(* Schneider Machine Expert - Basic project M221-KSB-single-pump, file version 2.0.0.0 *)
(* ProjectInformations: Name=KSB Single Pump Panel *)

HARDWARE
  Cpu 0: TM221CE24R
  ModuleExtensionObject 0: TM3TI4/G
  ModuleExtensionObject 1: TM3TI8T/G
  ModuleExtensionObject 2: TM3AI2H/G
  EthernetConfiguration: NetworkName=M221, IpAllocationMode=FixedAddress, IpAddress=192.168.1.107, SubnetMask=255.255.255.0
  SerialLineConfiguration: Baud=Baud19200, Parity=ParityEven, DataBits=DataBits8, StopBits=StopBits1, PhysicalMedium=PhysicalMediumRs485, TransmissionMode=TransmissionModeModbusRtu, SlaveId=1, Addressing=SlaveAddressing
  MastTask: UsePeriodScanMode=false, PeriodScan=100
  FastTask: Period=255
  CpuBehavior: StartingMode=StartInRun, AutoSaveRamOnEeprom=true, WatchdogPeriod=250

SYMBOLS  (address, symbol, comment, settings)
  %M0       SET_PLC_TIME  "Setting this bit allows you to change the PLC Time; gets set on negative transition of bit"
  %M1       SEAL_FAIL_ALARM
  %M2       HIGH_FLOAT_ALARM
  %M3       HIGH_VIBRATION_ALARM
  %M4       HIGH_BOTTOM_BEARING_TEMP_ALARM
  %M5       RESET_ALARMS
  %M6       SILENCE_ALARMS
  %M7       WINDING_TEMP_ALARM_BYPASS
  %M8       SEAL_FAIL_ALARM_BYPASS
  %M9       HIGH_FLOAT_ALARM_BYPASS
  %M10      VIBRATION_ALARM_BYPASS
  %M11      HIGH_BOT_BEAR_TMP_ALARM_BYPASS
  %M12      MODULE_1_STATUS
  %M13      MODULE_2_STATUS
  %M14      MODULE_3_STATUS
  %M110     LOGGING_DONE
  %M111     LOGGING_BUSY
  %M112     LOGGING_ERROR
  %M113     LOGGING_BAK
  %M114     LOG_NEXT
  %S6       SB_TB1S  "Time base of 1 s generated by an internal clock"
  %S13      SB_FIRSTRUN  "Indicates the first controller cycle in RUN mode"
  %S50      SB_RTCUPDATE  "Set to 1, this bit allows to update the date and time"
  %SW51     SW_RTCHHMM  "RTC Function: contains in BCD HHMM: hour and minute"
  %SW52     SW_RTCMMDD  "RTC Function: contains in BCD MMDD: month and day"
  %SW53     SW_RTCCCYY  "RTC Function: contains in BCD CCYY: century and year"
  %SW120    SW_IOSTATUS  "Shows expansion I/O module status (refer F1 help for details)"
  %MW0      DAY
  %MW1      HOUR  "My_Time"
  %MW2      MINUTES
  %MW3      MONTH
  %MW4      YEAR
  %MW5      SCRAP_MONTH  "Interim Register to Load into BCD"
  %MW6      SCRAP_MINUTES  "Interim Register to Load into BCD"
  %MW7      SEAL_FAIL_ALARM_DELAY_PRESET
  %MW8      VIBRATION_ALARM_DELAY_PRESET
  %MW9      WINDING1_TEMP_LOG
  %MW10     WINDING2_TEMP_LOG
  %MW11     WINDING3_TEMP_LOG
  %MW12     BOTTOM_BEARING_TEMP_LOG
  %MW13     WINDING_TEMP_LOG
  %MW14     VIBRATION_LOG
  %KW0      DISCONNECTED_VALUE  [Value=-32768]
  %TM0      HIGH_BOT_BEARING_TMP_ALARM_DELAY  [Preset=10, Base=OneSecond]
  %TM1      HIGH_FLOAT_ALARM_DELAY  [Preset=10, Base=OneSecond]
  %TM2      HIGH_WINDING_TEMP_ALARM_DELAY  [Preset=10, Base=OneSecond]
  %TM3      SEAL_FAIL_ALARM_DELAY  [Preset=10, Base=OneSecond]
  %TM4      VIBRATION_ALARM_DELAY  [Preset=10, Base=OneSecond]
  %TM5      NEXT_LOG_DELAY_TIMER  [Preset=30, Base=OneSecond]
  %DATALOG0   [Records(DataLoggingRecord(Value=%I0.0), DataLoggingRecord(Value=%IW1.0), DataLoggingRecord(Value=%IW1.1), DataLoggingRecord(Value=%IW1.2), DataLoggingRecord(Value=%IW1.3), DataLoggingRecord(Value=%IW2.0), DataLoggingRecord(Value=%IW3.0)), AddDateTime=true, DataLoggingType=HistoricalData, MaxFileSize=100]
  %DATALOG1   [Records(DataLoggingRecord(Value=%IW1.0)), AddDateTime=true, DataLoggingType=HistoricalData, MaxFileSize=500]
  %I0.0     SEAL_FAIL  "Reversed Logic Sensor!!! Normally Closed. Seal failing breaks connection"
  %I0.1     HIGH_FLOAT
  %Q0.0     PUMP_ENABLE
  %Q0.1     AUDIBLE_ALARM
  %IW1.0    WINDING1_TEMP  [Type=Type_PT100, Scope=Scope_Fahrenheit, Minimum=-3280, Maximum=15620]
  %IW1.1    WINDING2_TEMP  [Type=Type_PT100, Scope=Scope_Fahrenheit, Minimum=-3280, Maximum=15620]
  %IW1.2    WINDING3_TEMP  [Type=Type_PT100, Scope=Scope_Fahrenheit, Minimum=-3280, Maximum=15620]
  %IW1.3    BOTTOM_BEARING_TEMP  [Type=Type_PT100, Scope=Scope_Fahrenheit, Minimum=-3280, Maximum=15620]
  %IW2.0    WINDING_TEMP  [Type=Type_NTC, Scope=Scope_Fahrenheit, Minimum=-514, Maximum=1104]
  %IW3.0    VIBRATION  [Type=Type_4_20mA, Scope=Scope_Customized, Minimum=0, Maximum=10000]

POU Alarm Conditions
  (* SectionNumber=1 *)

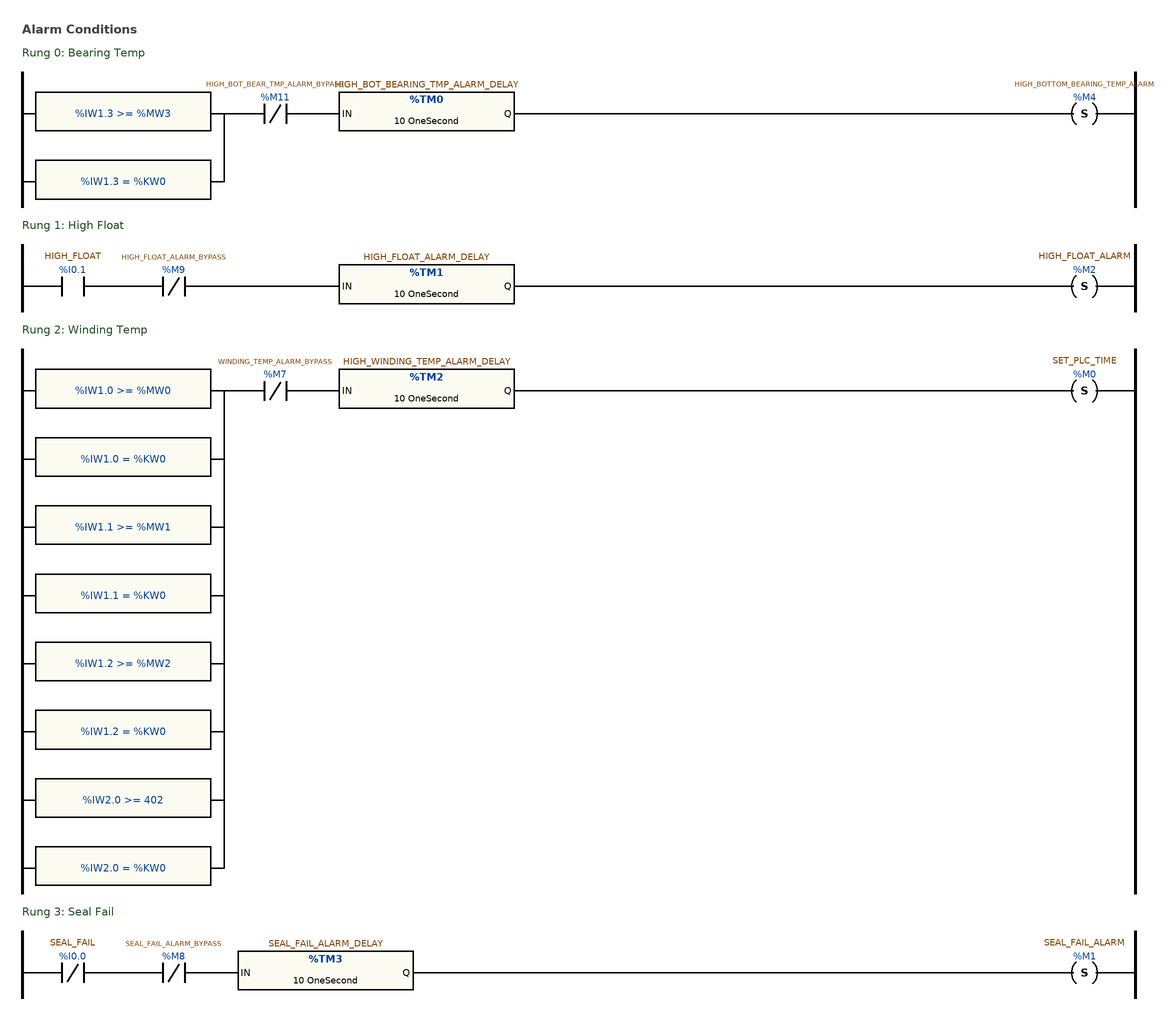

// Rung 0: Bearing Temp
  BLK %TM0                (* HIGH_BOT_BEARING_TMP_ALARM_DELAY *)
  LD [ %IW1.3 >= %MW3 ]   (* BOTTOM_BEARING_TEMP, MONTH *)
  OR [ %IW1.3 = %KW0 ]    (* BOTTOM_BEARING_TEMP, DISCONNECTED_VALUE *)
  ANDN %M11               (* HIGH_BOT_BEAR_TMP_ALARM_BYPASS *)
  IN
  OUT_BLK
  LD Q
  S %M4                   (* HIGH_BOTTOM_BEARING_TEMP_ALARM *)
  END_BLK
  // as ST:
  //   HIGH_BOT_BEARING_TMP_ALARM_DELAY(IN := (BOTTOM_BEARING_TEMP >= MONTH OR BOTTOM_BEARING_TEMP = DISCONNECTED_VALUE) AND NOT HIGH_BOT_BEAR_TMP_ALARM_BYPASS);
  //   IF HIGH_BOT_BEARING_TMP_ALARM_DELAY.Q THEN HIGH_BOTTOM_BEARING_TEMP_ALARM := TRUE; END_IF;

// Rung 1: High Float
  BLK %TM1                (* HIGH_FLOAT_ALARM_DELAY *)
  LD %I0.1                (* HIGH_FLOAT *)
  ANDN %M9                (* HIGH_FLOAT_ALARM_BYPASS *)
  IN
  OUT_BLK
  LD Q
  S %M2                   (* HIGH_FLOAT_ALARM *)
  END_BLK
  // as ST:
  //   HIGH_FLOAT_ALARM_DELAY(IN := HIGH_FLOAT AND NOT HIGH_FLOAT_ALARM_BYPASS);
  //   IF HIGH_FLOAT_ALARM_DELAY.Q THEN HIGH_FLOAT_ALARM := TRUE; END_IF;

// Rung 2: Winding Temp
  BLK %TM2                (* HIGH_WINDING_TEMP_ALARM_DELAY *)
  LD [ %IW1.0 >= %MW0 ]   (* WINDING1_TEMP, DAY *)
  OR [ %IW1.0 = %KW0 ]    (* WINDING1_TEMP, DISCONNECTED_VALUE *)
  OR [ %IW1.1 >= %MW1 ]   (* WINDING2_TEMP, HOUR *)
  OR [ %IW1.1 = %KW0 ]    (* WINDING2_TEMP, DISCONNECTED_VALUE *)
  OR [ %IW1.2 >= %MW2 ]   (* WINDING3_TEMP, MINUTES *)
  OR [ %IW1.2 = %KW0 ]    (* WINDING3_TEMP, DISCONNECTED_VALUE *)
  OR [ %IW2.0 >= 402 ]    (* WINDING_TEMP *)
  OR [ %IW2.0 = %KW0 ]    (* WINDING_TEMP, DISCONNECTED_VALUE *)
  ANDN %M7                (* WINDING_TEMP_ALARM_BYPASS *)
  IN
  OUT_BLK
  LD Q
  S %M0                   (* SET_PLC_TIME *)
  END_BLK
  // as ST:
  //   HIGH_WINDING_TEMP_ALARM_DELAY(IN := (WINDING1_TEMP >= DAY OR WINDING1_TEMP = DISCONNECTED_VALUE OR WINDING2_TEMP >= HOUR OR WINDING2_TEMP = DISCONNECTED_VALUE OR WINDING3_TEMP >= MINUTES OR WINDING3_TEMP = DISCONNECTED_VALUE OR WINDING_TEMP >= 402 OR WINDING_TEMP = DISCONNECTED_VALUE) AND NOT WINDING_TEMP_ALARM_BYPASS);
  //   IF HIGH_WINDING_TEMP_ALARM_DELAY.Q THEN SET_PLC_TIME := TRUE; END_IF;

// Rung 3: Seal Fail
  BLK %TM3                (* SEAL_FAIL_ALARM_DELAY *)
  LDN %I0.0               (* SEAL_FAIL *)
  ANDN %M8                (* SEAL_FAIL_ALARM_BYPASS *)
  IN
  OUT_BLK
  LD Q
  S %M1                   (* SEAL_FAIL_ALARM *)
  END_BLK
  // as ST:
  //   SEAL_FAIL_ALARM_DELAY(IN := NOT SEAL_FAIL AND NOT SEAL_FAIL_ALARM_BYPASS);
  //   IF SEAL_FAIL_ALARM_DELAY.Q THEN SEAL_FAIL_ALARM := TRUE; END_IF;

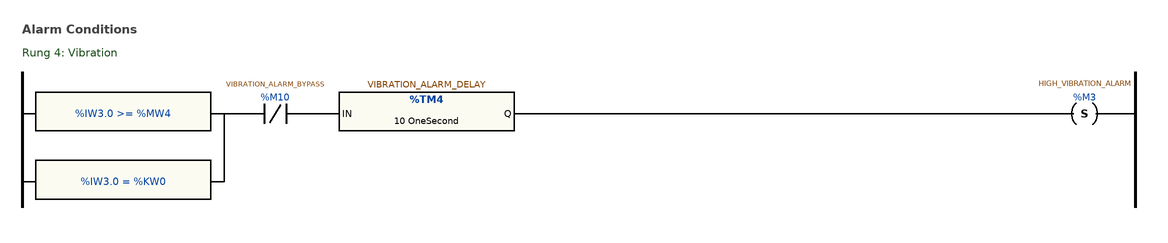

// Rung 4: Vibration
  BLK %TM4                (* VIBRATION_ALARM_DELAY *)
  LD [ %IW3.0 >= %MW4 ]   (* VIBRATION, YEAR *)
  OR [ %IW3.0 = %KW0 ]    (* VIBRATION, DISCONNECTED_VALUE *)
  ANDN %M10               (* VIBRATION_ALARM_BYPASS *)
  IN
  OUT_BLK
  LD Q
  S %M3                   (* HIGH_VIBRATION_ALARM *)
  END_BLK
  // as ST:
  //   VIBRATION_ALARM_DELAY(IN := (VIBRATION >= YEAR OR VIBRATION = DISCONNECTED_VALUE) AND NOT VIBRATION_ALARM_BYPASS);
  //   IF VIBRATION_ALARM_DELAY.Q THEN HIGH_VIBRATION_ALARM := TRUE; END_IF;

POU Pump Enable
  (* SectionNumber=2 *)

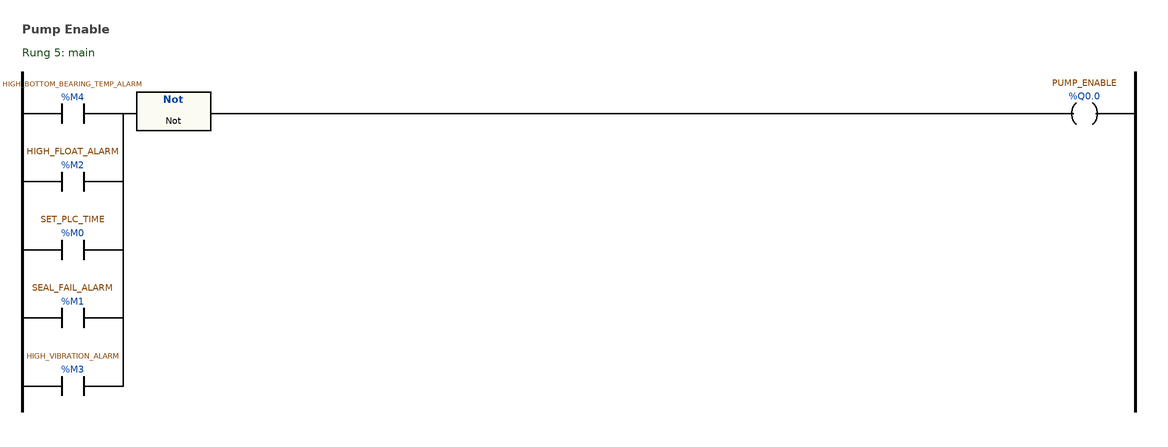

// Rung 5: main
  LD %M4                  (* HIGH_BOTTOM_BEARING_TEMP_ALARM *)
  OR %M2                  (* HIGH_FLOAT_ALARM *)
  OR %M0                  (* SET_PLC_TIME *)
  OR %M1                  (* SEAL_FAIL_ALARM *)
  OR %M3                  (* HIGH_VIBRATION_ALARM *)
  N
  ST %Q0.0                (* PUMP_ENABLE *)
  // as ST:
  //   PUMP_ENABLE := NOT (HIGH_BOTTOM_BEARING_TEMP_ALARM OR HIGH_FLOAT_ALARM OR SET_PLC_TIME OR SEAL_FAIL_ALARM OR HIGH_VIBRATION_ALARM);

POU Resets
  (* SectionNumber=3 *)

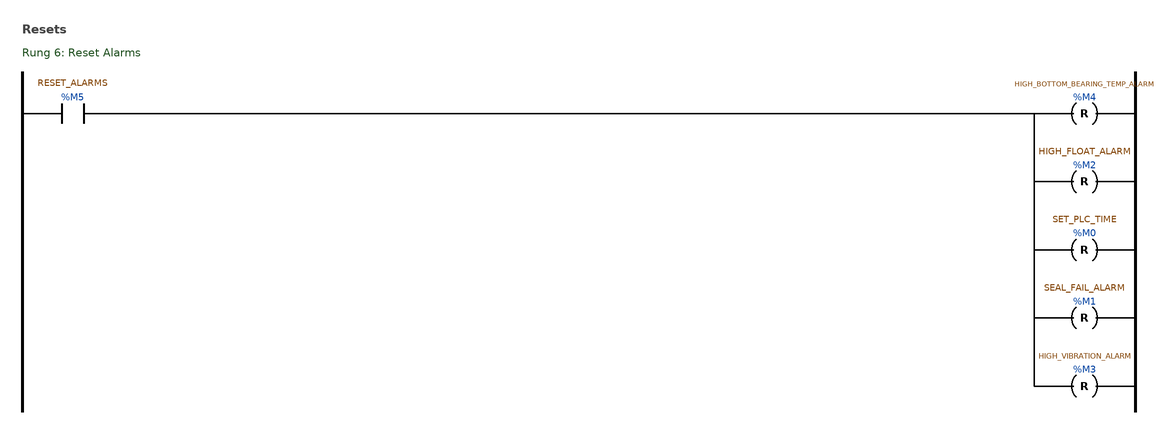

// Rung 6: Reset Alarms
  LD %M5                  (* RESET_ALARMS *)
  R %M4                   (* HIGH_BOTTOM_BEARING_TEMP_ALARM *)
  R %M2                   (* HIGH_FLOAT_ALARM *)
  R %M0                   (* SET_PLC_TIME *)
  R %M1                   (* SEAL_FAIL_ALARM *)
  R %M3                   (* HIGH_VIBRATION_ALARM *)
  // as ST:
  //   IF RESET_ALARMS THEN HIGH_BOTTOM_BEARING_TEMP_ALARM := FALSE; END_IF;
  //   IF RESET_ALARMS THEN HIGH_FLOAT_ALARM := FALSE; END_IF;
  //   IF RESET_ALARMS THEN SET_PLC_TIME := FALSE; END_IF;
  //   IF RESET_ALARMS THEN SEAL_FAIL_ALARM := FALSE; END_IF;
  //   IF RESET_ALARMS THEN HIGH_VIBRATION_ALARM := FALSE; END_IF;

POU On Startup
  (* SectionNumber=4 *)

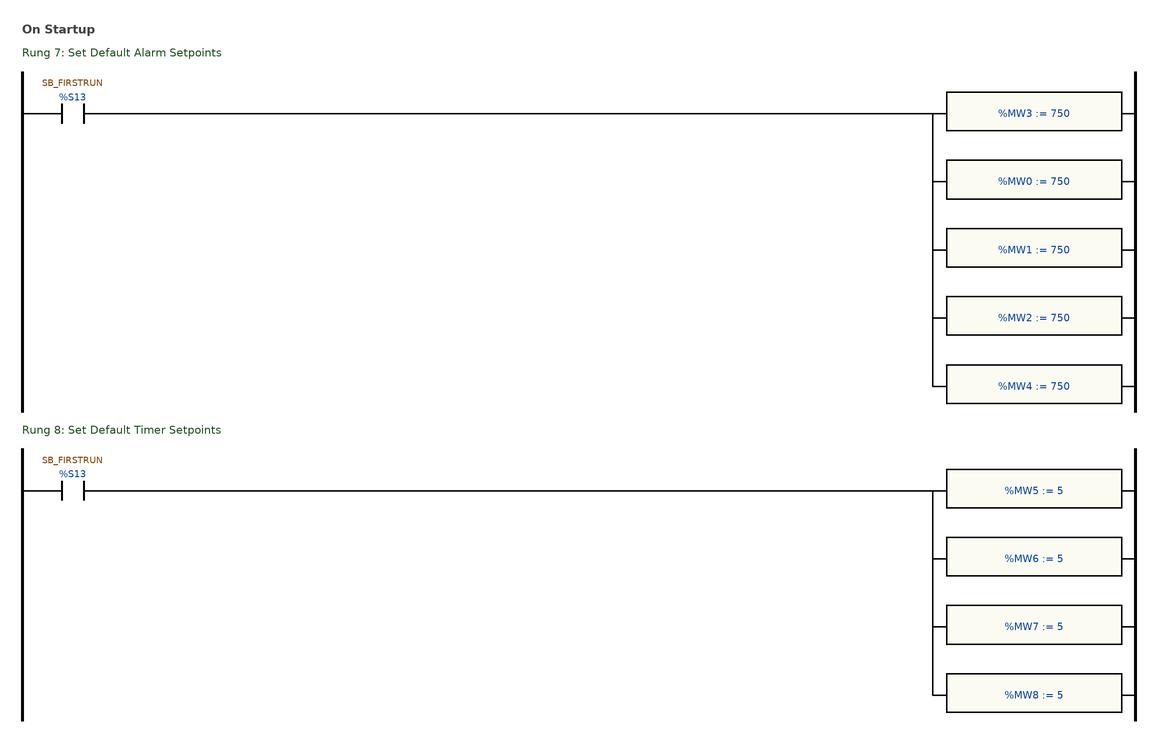

// Rung 7: Set Default Alarm Setpoints
  LD %S13                 (* SB_FIRSTRUN *)
  [ %MW3 := 750 ]         (* MONTH *)
  [ %MW0 := 750 ]         (* DAY *)
  [ %MW1 := 750 ]         (* HOUR *)
  [ %MW2 := 750 ]         (* MINUTES *)
  [ %MW4 := 750 ]         (* YEAR *)
  // as ST:
  //   IF SB_FIRSTRUN THEN MONTH := 750; END_IF;
  //   IF SB_FIRSTRUN THEN DAY := 750; END_IF;
  //   IF SB_FIRSTRUN THEN HOUR := 750; END_IF;
  //   IF SB_FIRSTRUN THEN MINUTES := 750; END_IF;
  //   IF SB_FIRSTRUN THEN YEAR := 750; END_IF;

// Rung 8: Set Default Timer Setpoints
  LD %S13                 (* SB_FIRSTRUN *)
  [ %MW5 := 5 ]           (* SCRAP_MONTH *)
  [ %MW6 := 5 ]           (* SCRAP_MINUTES *)
  [ %MW7 := 5 ]           (* SEAL_FAIL_ALARM_DELAY_PRESET *)
  [ %MW8 := 5 ]           (* VIBRATION_ALARM_DELAY_PRESET *)
  // as ST:
  //   IF SB_FIRSTRUN THEN SCRAP_MONTH := 5; END_IF;
  //   IF SB_FIRSTRUN THEN SCRAP_MINUTES := 5; END_IF;
  //   IF SB_FIRSTRUN THEN SEAL_FAIL_ALARM_DELAY_PRESET := 5; END_IF;
  //   IF SB_FIRSTRUN THEN VIBRATION_ALARM_DELAY_PRESET := 5; END_IF;

POU Timers
  (* SectionNumber=5 *)

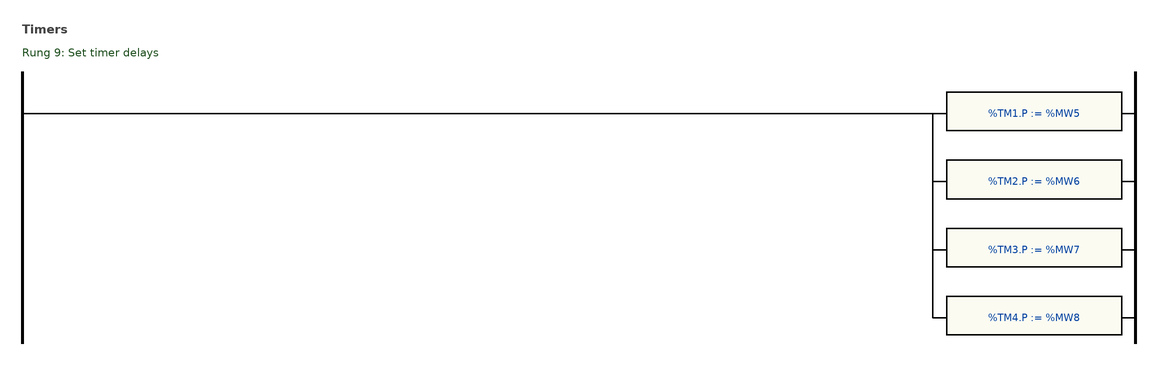

// Rung 9: Set timer delays
  LD 1
  [ %TM1.P := %MW5 ]      (* HIGH_FLOAT_ALARM_DELAY, SCRAP_MONTH *)
  [ %TM2.P := %MW6 ]      (* HIGH_WINDING_TEMP_ALARM_DELAY, SCRAP_MINUTES *)
  [ %TM3.P := %MW7 ]      (* SEAL_FAIL_ALARM_DELAY, SEAL_FAIL_ALARM_DELAY_PRESET *)
  [ %TM4.P := %MW8 ]      (* VIBRATION_ALARM_DELAY, VIBRATION_ALARM_DELAY_PRESET *)
  // as ST:
  //   HIGH_FLOAT_ALARM_DELAY.P := SCRAP_MONTH;
  //   HIGH_WINDING_TEMP_ALARM_DELAY.P := SCRAP_MINUTES;
  //   SEAL_FAIL_ALARM_DELAY.P := SEAL_FAIL_ALARM_DELAY_PRESET;
  //   VIBRATION_ALARM_DELAY.P := VIBRATION_ALARM_DELAY_PRESET;

POU Logging Variables
  (* SectionNumber=6 *)

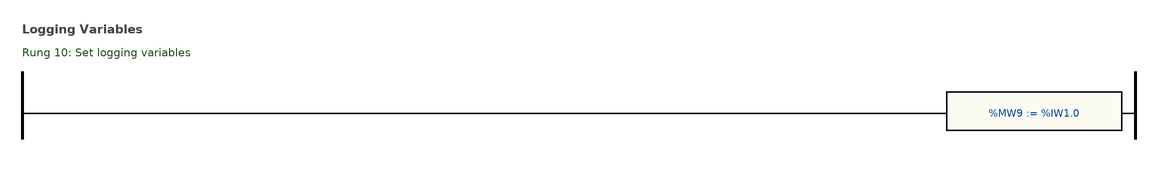

// Rung 10: Set logging variables
  LD 1
  [ %MW9 := %IW1.0 ]      (* WINDING1_TEMP_LOG, WINDING1_TEMP *)
  // as ST:
  //   WINDING1_TEMP_LOG := WINDING1_TEMP;

POU DataLogger
  (* SectionNumber=7 *)

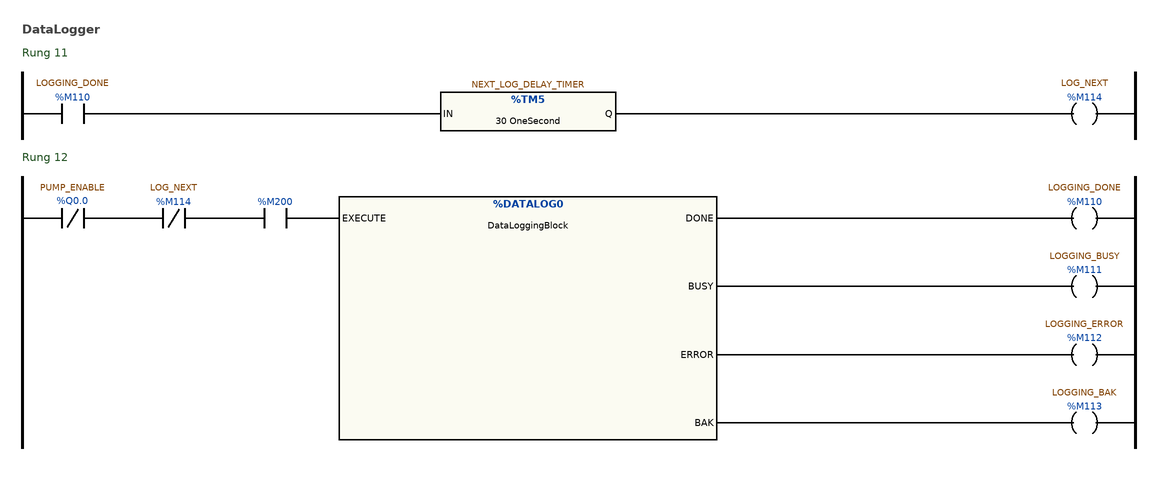

// Rung 11
  BLK %TM5                (* NEXT_LOG_DELAY_TIMER *)
  LD %M110                (* LOGGING_DONE *)
  IN
  OUT_BLK
  LD Q
  ST %M114                (* LOG_NEXT *)
  END_BLK
  // as ST:
  //   NEXT_LOG_DELAY_TIMER(IN := LOGGING_DONE);
  //   LOG_NEXT := NEXT_LOG_DELAY_TIMER.Q;

// Rung 12
  BLK %DATALOG0
  LDN %Q0.0               (* PUMP_ENABLE *)
  ANDN %M114              (* LOG_NEXT *)
  AND %M200
  EXECUTE
  OUT_BLK
  LD DONE
  ST %M110                (* LOGGING_DONE *)
  LD BUSY
  ST %M111                (* LOGGING_BUSY *)
  LD ERROR
  ST %M112                (* LOGGING_ERROR *)
  LD BAK
  ST %M113                (* LOGGING_BAK *)
  END_BLK
  // as ST:
  //   %DATALOG0(EXECUTE := NOT PUMP_ENABLE AND NOT LOG_NEXT AND %M200);
  //   LOGGING_DONE := %DATALOG0.DONE;
  //   LOGGING_BUSY := %DATALOG0.BUSY;
  //   LOGGING_ERROR := %DATALOG0.ERROR;
  //   LOGGING_BAK := %DATALOG0.BAK;

POU DataLogger_Test
  (* SectionNumber=8 *)

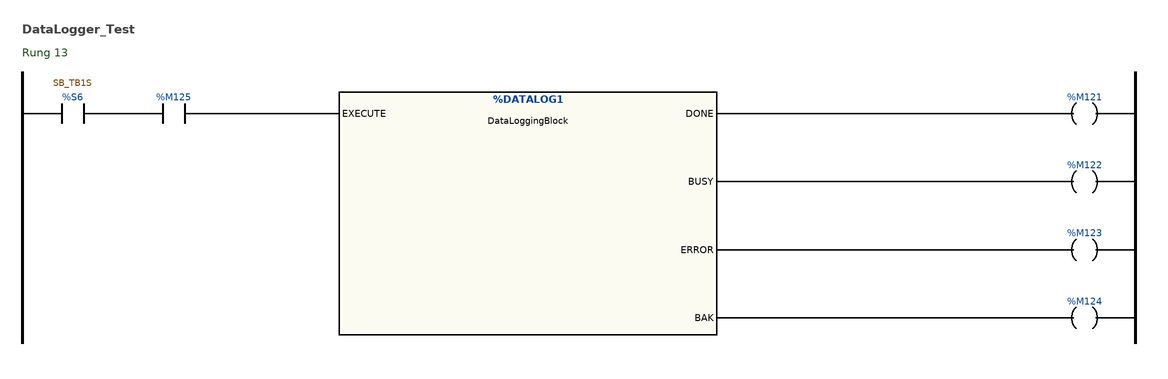

// Rung 13
  BLK %DATALOG1
  LD %S6                  (* SB_TB1S *)
  AND %M125
  EXECUTE
  OUT_BLK
  LD DONE
  ST %M121
  LD BUSY
  ST %M122
  LD ERROR
  ST %M123
  LD BAK
  ST %M124
  END_BLK
  // as ST:
  //   %DATALOG1(EXECUTE := SB_TB1S AND %M125);
  //   %M121 := %DATALOG1.DONE;
  //   %M122 := %DATALOG1.BUSY;
  //   %M123 := %DATALOG1.ERROR;
  //   %M124 := %DATALOG1.BAK;

POU ModuleStatus
  (* SectionNumber=9 *)

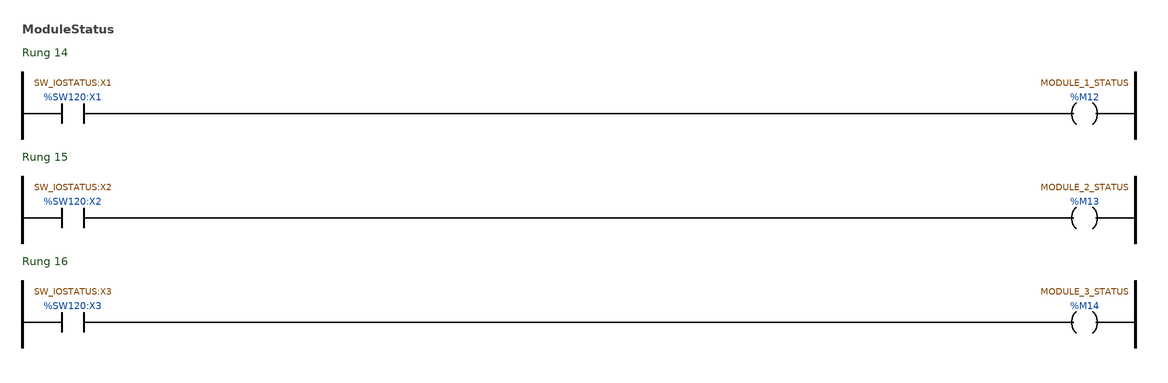

// Rung 14
  LD %SW120:X1            (* SW_IOSTATUS *)
  ST %M12                 (* MODULE_1_STATUS *)
  // as ST:
  //   MODULE_1_STATUS := SW_IOSTATUS:X1;

// Rung 15
  LD %SW120:X2            (* SW_IOSTATUS *)
  ST %M13                 (* MODULE_2_STATUS *)
  // as ST:
  //   MODULE_2_STATUS := SW_IOSTATUS:X2;

// Rung 16
  LD %SW120:X3            (* SW_IOSTATUS *)
  ST %M14                 (* MODULE_3_STATUS *)
  // as ST:
  //   MODULE_3_STATUS := SW_IOSTATUS:X3;

POU PLC Time to HMI
  (* SectionNumber=1 *)

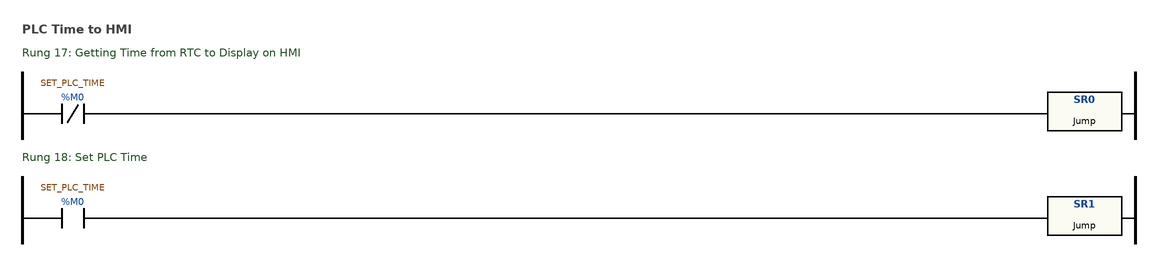

// Rung 17: Getting Time from RTC to Display on HMI
  LDN %M0                 (* SET_PLC_TIME *)
  SR0
  // as ST:
  //   IF NOT SET_PLC_TIME THEN SR0(); END_IF;

// Rung 18: Set PLC Time
  LD %M0                  (* SET_PLC_TIME *)
  SR1
  // as ST:
  //   IF SET_PLC_TIME THEN SR1(); END_IF;

Subroutine Get RTC
  (* SectionNumber=2, Number=0 *)

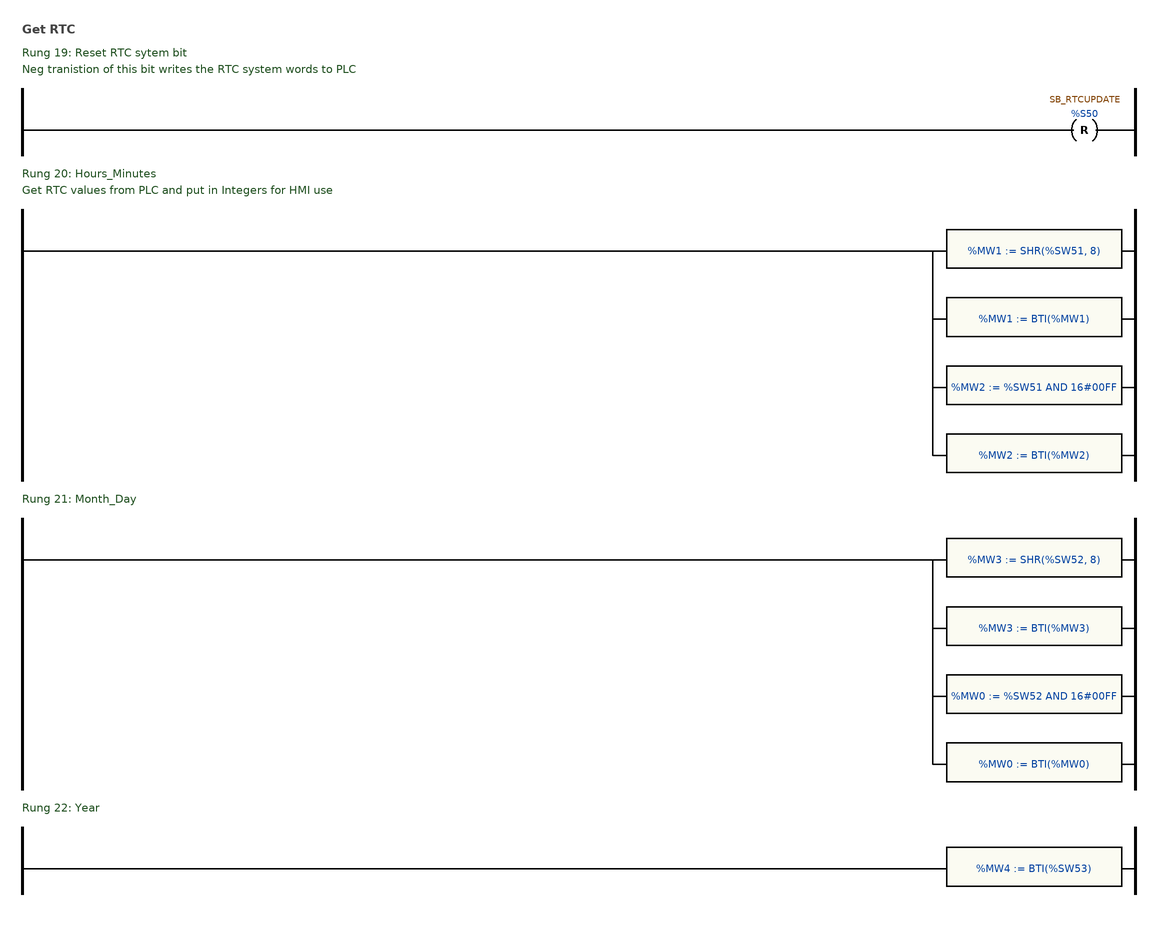

// Rung 19: Reset RTC sytem bit
// Neg tranistion of this bit writes the RTC system words to PLC
  LD 1
  R %S50                  (* SB_RTCUPDATE *)
  // as ST:
  //   SB_RTCUPDATE := FALSE;

// Rung 20: Hours_Minutes
// Get RTC values from PLC and put in Integers for HMI use
  LD 1
  [ %MW1 := SHR ( %SW51 , 8 ) ](* HOUR, SW_RTCHHMM *)
  [ %MW1 := BTI ( %MW1 ) ](* HOUR, HOUR *)
  [ %MW2 := %SW51 AND 16#00FF ](* MINUTES, SW_RTCHHMM *)
  [ %MW2 := BTI ( %MW2 ) ](* MINUTES, MINUTES *)
  // as ST:
  //   HOUR := SHR ( SW_RTCHHMM , 8 );
  //   HOUR := BTI ( HOUR );
  //   MINUTES := SW_RTCHHMM AND 16#00FF;
  //   MINUTES := BTI ( MINUTES );

// Rung 21: Month_Day
  LD 1
  [ %MW3 := SHR ( %SW52 , 8 ) ](* MONTH, SW_RTCMMDD *)
  [ %MW3 := BTI ( %MW3 ) ](* MONTH, MONTH *)
  [ %MW0 := %SW52 AND 16#00FF ](* DAY, SW_RTCMMDD *)
  [ %MW0 := BTI ( %MW0 ) ](* DAY, DAY *)
  // as ST:
  //   MONTH := SHR ( SW_RTCMMDD , 8 );
  //   MONTH := BTI ( MONTH );
  //   DAY := SW_RTCMMDD AND 16#00FF;
  //   DAY := BTI ( DAY );

// Rung 22: Year
  LD 1
  [%MW4 := BTI(%SW53)]    (* YEAR, SW_RTCCCYY *)
  // as ST:
  //   YEAR := BTI(SW_RTCCCYY);

Subroutine Set RTC
  (* SectionNumber=3, Number=1 *)

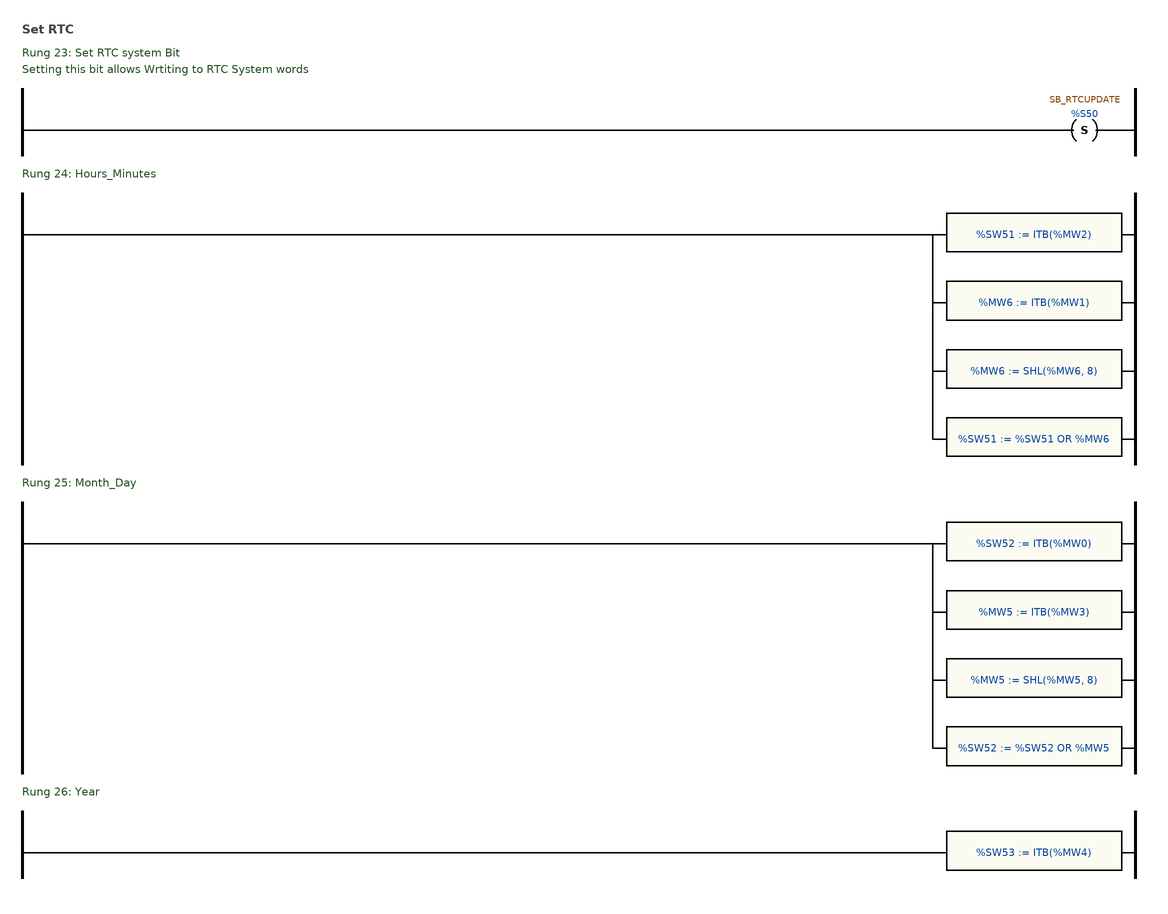

// Rung 23: Set RTC system Bit
// Setting this bit allows Wrtiting to RTC System words
  LD 1
  S %S50                  (* SB_RTCUPDATE *)
  // as ST:
  //   SB_RTCUPDATE := TRUE;

// Rung 24: Hours_Minutes
  LD 1
  [%SW51 := ITB(%MW2)]    (* SW_RTCHHMM, MINUTES *)
  [%MW6 := ITB(%MW1)]     (* SCRAP_MINUTES, HOUR *)
  [%MW6 := SHL(%MW6, 8)]  (* SCRAP_MINUTES, SCRAP_MINUTES *)
  [%SW51 := %SW51 OR %MW6](* SW_RTCHHMM, SW_RTCHHMM, SCRAP_MINUTES *)
  // as ST:
  //   SW_RTCHHMM := ITB(MINUTES);
  //   SCRAP_MINUTES := ITB(HOUR);
  //   SCRAP_MINUTES := SHL(SCRAP_MINUTES, 8);
  //   SW_RTCHHMM := SW_RTCHHMM OR SCRAP_MINUTES;

// Rung 25: Month_Day
  LD 1
  [%SW52 := ITB(%MW0)]    (* SW_RTCMMDD, DAY *)
  [%MW5 := ITB(%MW3)]     (* SCRAP_MONTH, MONTH *)
  [%MW5 := SHL(%MW5, 8)]  (* SCRAP_MONTH, SCRAP_MONTH *)
  [%SW52 := %SW52 OR %MW5](* SW_RTCMMDD, SW_RTCMMDD, SCRAP_MONTH *)
  // as ST:
  //   SW_RTCMMDD := ITB(DAY);
  //   SCRAP_MONTH := ITB(MONTH);
  //   SCRAP_MONTH := SHL(SCRAP_MONTH, 8);
  //   SW_RTCMMDD := SW_RTCMMDD OR SCRAP_MONTH;

// Rung 26: Year
  LD 1
  [%SW53 := ITB(%MW4)]    (* SW_RTCCCYY, YEAR *)
  // as ST:
  //   SW_RTCCCYY := ITB(YEAR);
